FUNCTION WithinRange : BOOL
VAR_INPUT
	ValA	:	REAL; //New position to evaluate
	Center :	REAL; //Current position
	Range : REAL; //Span of the range
	Offset	:	REAL := 0; //Offset from center if the range is non-symetric
END_VAR
VAR
END_VAR

IF ValA < (Center + Offset - (Range/2) ) THEN
	WithinRange := FALSE;
ELSIF ValA > (Center + Offset + (Range/2) ) THEN
	WithinRange := FALSE;
ELSE
	WithinRange := TRUE;
END_IF

END_FUNCTION

(* stored: Version 1.1.0.1, ProductVersion 3.1.4020.12
   POU WithinRange: Id {4bb5698f-fd10-4025-99c8-626222c4591f}, SpecialFunc None *)
